(* IEC 61131-3 sources: plc_generation_empirical_study/datasets/task_bank_v0_3/tasks/C04_B13_composite, 2 files *)

(* ---- interface.st ---- *)
FUNCTION_BLOCK C04_B13_composite
VAR_INPUT
    A_Button : BOOL;
    A_Enable : BOOL;
    A_Reset : BOOL;
    B_Event : BOOL;
    B_Qualify : BOOL;
    B_Reset : BOOL;
    B_MaxCount : INT;
    SubsystemBEnable : BOOL;
    CrossReset : BOOL;
END_VAR
VAR_OUTPUT
    A_State : BOOL;
    A_AcceptedPulse : BOOL;
    B_Count : INT;
    B_AcceptedPulse : BOOL;
    B_AtLimit : BOOL;
    CrossReady : BOOL;
    CrossBlocked : BOOL;
END_VAR
END_FUNCTION_BLOCK

(* ---- reference.st ---- *)
FUNCTION_BLOCK C04_B13_composite
VAR_INPUT
    A_Button : BOOL;
    A_Enable : BOOL;
    A_Reset : BOOL;
    B_Event : BOOL;
    B_Qualify : BOOL;
    B_Reset : BOOL;
    B_MaxCount : INT;
    SubsystemBEnable : BOOL;
    CrossReset : BOOL;
END_VAR
VAR_OUTPUT
    A_State : BOOL;
    A_AcceptedPulse : BOOL;
    B_Count : INT;
    B_AcceptedPulse : BOOL;
    B_AtLimit : BOOL;
    CrossReady : BOOL;
    CrossBlocked : BOOL;
END_VAR
VAR
    A_PrevButton : BOOL := FALSE;
    B_PrevEvent : BOOL := FALSE;
END_VAR

A_AcceptedPulse := FALSE;
IF A_Reset THEN
    A_State := FALSE;
ELSIF A_Enable AND A_Button AND (NOT A_PrevButton) THEN
    A_State := NOT A_State;
    A_AcceptedPulse := TRUE;
END_IF;
A_PrevButton := A_Button;

IF CrossReset THEN
    CrossReady := FALSE;
ELSIF A_State THEN
    CrossReady := TRUE;
END_IF;
CrossBlocked := SubsystemBEnable AND (NOT CrossReady);

IF SubsystemBEnable AND CrossReady THEN
    B_AcceptedPulse := FALSE;
    IF B_Reset THEN
        B_Count := 0;
    ELSIF B_Event AND (NOT B_PrevEvent) AND B_Qualify AND (B_Count < B_MaxCount) THEN
        B_Count := B_Count + 1;
        B_AcceptedPulse := TRUE;
    END_IF;
    B_AtLimit := B_Count >= B_MaxCount;
    B_PrevEvent := B_Event;
ELSE
    B_Count := 0;
    B_AcceptedPulse := FALSE;
    B_AtLimit := FALSE;
END_IF;

END_FUNCTION_BLOCK
